FUNCTION_BLOCK Machine EXTENDS FB_PackML_BaseModule
VAR
	RackAndPinion	: FB_RackAndPinion;
END_VAR

METHOD PROTECTED HMIPermissions
AllowHMIControl(TRUE);
END_METHOD

(* Basic module initialization logic*)
METHOD PROTECTED Initialize : BOOL
Initialize := FALSE;
CASE DescendantSequenceState OF
	0:
		RegisterSubmodule(SubModule := RackAndPinion);
		DescendantSequenceState := DescendantSequenceState + 10;

	10:
		IF SUPER^.Initialize() THEN
			Initialize := TRUE;
		END_IF
END_CASE
END_METHOD

END_FUNCTION_BLOCK

(* stored: Version 1.1.0.1
   POU Machine: Id {f6ae2cbe-173e-4d75-bb5e-334498954288}, SpecialFunc None
   Method HMIPermissions: Id {01f1aea6-e802-48f8-abd4-50a2a3d31fba}
   Method Initialize: Id {563069b4-df21-4c5b-a8db-0fb2d2934ac8} *)
